PROGRAM MAIN
VAR
	StopRichiesto: BOOL;
	Anomalia: BOOL;
	Emergenza: BOOL;
	Funzione: BOOL;
	Smistamento: BOOL;
	Rotazione: BOOL;
	AttivaMicroRulli: BOOL;
	FineSmistamento: BOOL;
	FinePesatura: BOOL;
	RuotaOrigine: BOOL;
	PesoMin5: BOOL;
	PesoMag10: BOOL;
	PesoIntermedio: BOOL;
	ProsciuttoSmistato: BOOL;
	//Timer
	TON_PS1: TON;
	TON_Pesatura: TON;
	TON_MicroRulli: TON;
END_VAR

GestionePulsanti();
GestioneMotori();
GestionePesatura();
GestioneRotazione();
GestioneSmistamento();

ACTION GestioneMotori:
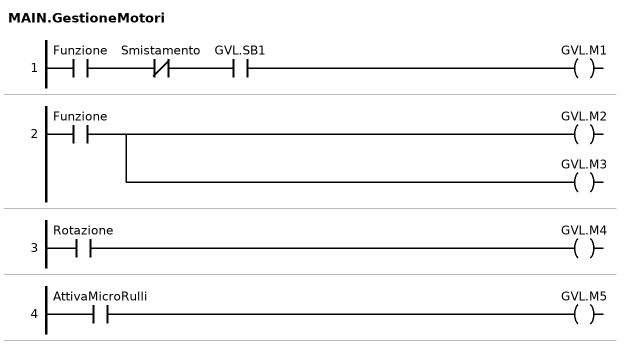
// NETWORK 1
GVL.M1 := Funzione AND NOT Smistamento AND GVL.SB1;

// NETWORK 2
GVL.M2 := Funzione;
GVL.M3 := Funzione;

// NETWORK 3
GVL.M4 := Rotazione;

// NETWORK 4
GVL.M5 := AttivaMicroRulli;
END_ACTION

ACTION GestionePesatura:
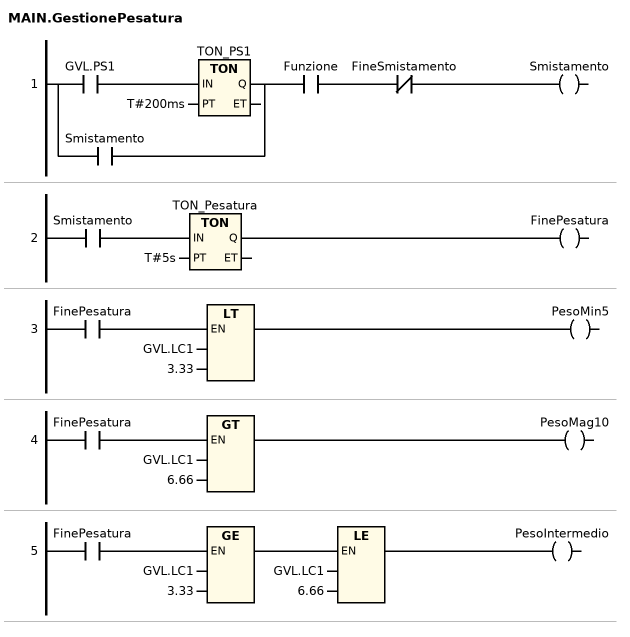
// NETWORK 1
TON_PS1(IN := GVL.PS1, PT := T#200ms); // TON
Smistamento := (TON_PS1.Q OR Smistamento) AND Funzione AND NOT FineSmistamento;

// NETWORK 2
TON_Pesatura(IN := Smistamento, PT := T#5s); // TON
FinePesatura := TON_Pesatura.Q;

// NETWORK 3
PesoMin5 := FinePesatura AND GVL.LC1 < 3.33;

// NETWORK 4
PesoMag10 := FinePesatura AND GVL.LC1 > 6.66;

// NETWORK 5
PesoIntermedio := FinePesatura AND GVL.LC1 >= 3.33 AND GVL.LC1 <= 6.66;
END_ACTION

ACTION GestionePulsanti:
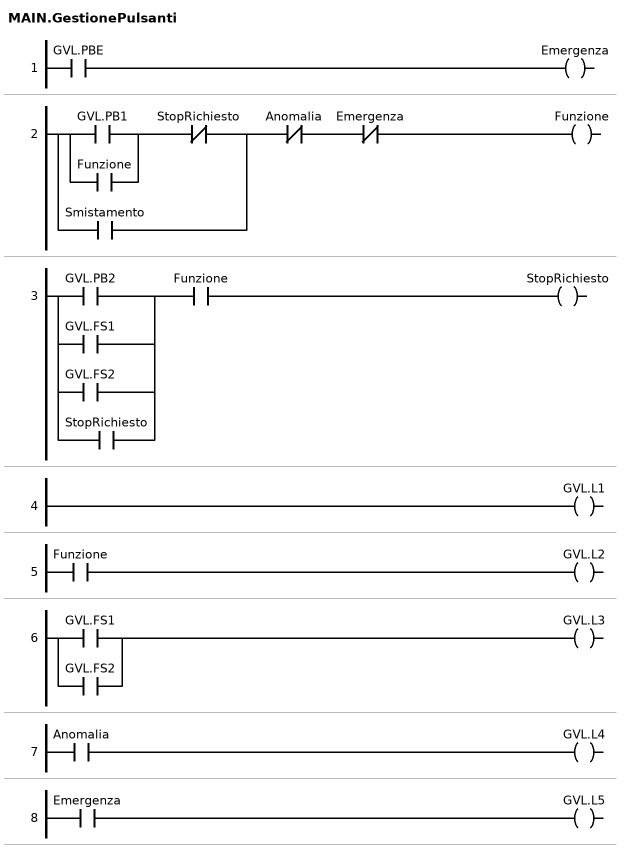
// NETWORK 1
Emergenza := GVL.PBE;

// NETWORK 2
Funzione := ((GVL.PB1 OR Funzione) AND NOT StopRichiesto OR Smistamento) AND NOT Anomalia AND NOT Emergenza;

// NETWORK 3
StopRichiesto := (GVL.PB2 OR GVL.FS1 OR GVL.FS2 OR StopRichiesto) AND Funzione;

// NETWORK 4
GVL.L1 := TRUE;

// NETWORK 5
GVL.L2 := Funzione;

// NETWORK 6
GVL.L3 := GVL.FS1 OR GVL.FS2;

// NETWORK 7
GVL.L4 := Anomalia;

// NETWORK 8
GVL.L5 := Emergenza;
END_ACTION

ACTION GestioneRotazione:
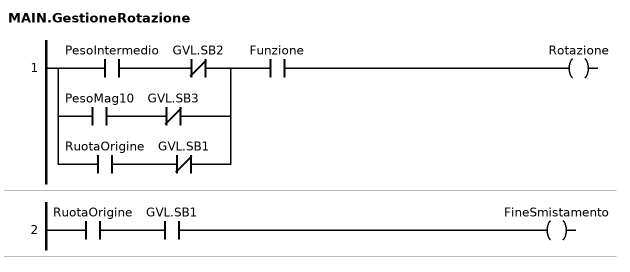
// NETWORK 1
Rotazione := (PesoIntermedio AND NOT GVL.SB2 OR PesoMag10 AND NOT GVL.SB3 OR RuotaOrigine AND NOT GVL.SB1) AND Funzione;

// NETWORK 2
FineSmistamento := RuotaOrigine AND GVL.SB1;
END_ACTION

ACTION GestioneSmistamento:
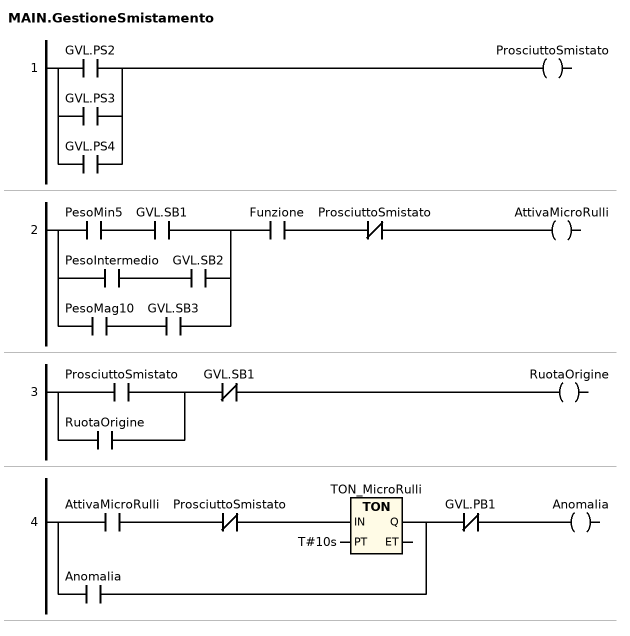
// NETWORK 1
ProsciuttoSmistato := GVL.PS2 OR GVL.PS3 OR GVL.PS4;

// NETWORK 2
AttivaMicroRulli := (PesoMin5 AND GVL.SB1 OR PesoIntermedio AND GVL.SB2 OR PesoMag10 AND GVL.SB3) AND Funzione AND NOT ProsciuttoSmistato;

// NETWORK 3
RuotaOrigine := (ProsciuttoSmistato OR RuotaOrigine) AND NOT GVL.SB1;

// NETWORK 4
TON_MicroRulli(IN := AttivaMicroRulli AND NOT ProsciuttoSmistato, PT := T#10s); // TON
Anomalia := (TON_MicroRulli.Q OR Anomalia) AND NOT GVL.PB1;
END_ACTION

END_PROGRAM

(* stored: Version 1.1.0.1, ProductVersion 3.1.4024.12
   POU MAIN: Id {77ce3c58-9155-42f5-9eb6-c02febfddbf9}, SpecialFunc None
   Action GestioneMotori: Id {90fd2a52-73a3-4857-abe4-70f7165621aa}
   Action GestionePesatura: Id {afcac87d-3588-48ef-84da-e3c3b38ed934}
   Action GestionePulsanti: Id {3f00a759-f8d0-455e-af78-03f29b3994ec}
   Action GestioneRotazione: Id {dcd47c17-31b5-470b-b8df-fa6a694df16f}
   Action GestioneSmistamento: Id {6af05be5-420f-47a5-a7ce-bdc4d670b5af} *)
